PROGRAM PRG_SampleState
VAR
	fbStateMachine			:FB_StateMachine;
	sCurrentState			:STRING;
	bBtnStart				:BOOL;
	bBtnStop				:BOOL;
	bError					:BOOL;
END_VAR

fbStateMachine(
				in_bError	:= bError, 
				in_bStart	:= bBtnStart, 
				in_bStop	:= bBtnStop, 
				out_ipState	=> );

sCurrentState := fbStateMachine.out_ipState.CurrentState;

END_PROGRAM

(* stored: Version 1.1.0.1
   POU PRG_SampleState: Id {07367209-6c29-4bd0-b647-9c5ae74e8c7f}, SpecialFunc None *)
